(* IEC 61131-3 sources: SafePLC-Gen-Evaluation/Evaluation Results/Dexpi_PDF/run_01, 2 files *)

(* ---- io_declarations.st ---- *)
(* ==================================================  *)
(* PLC I/O Variable Declarations — CODESYS 3.5  *)
(* Generated by SafePLC-Gen Multimodal  *)
(* ==================================================  *)

VAR_GLOBAL
    (* --- Analog Inputs ---  *)
    PI_4712.01_Raw               AT %IW0       : INT := 0;    (* PI-4712.01 — Pressure indicator, local, on process li  *)
    PICSA_4712.02_Raw            AT %IW2       : INT := 0;    (* PICSA-4712.02 — Pressure indicator, controller, switch,   *)
    TICSA_4750.03_Raw            AT %IW4       : INT := 0;    (* TICSA-4750.03 — Temperature indicator, controller, switc  *)
    (* --- Analog Outputs ---  *)
    MV_73KH12_25_Out             AT %QW0       : INT := 0;    (* MV-73KH12-25 — Manual isolation valve on line 73KH12-25  *)
    MV_73KH12_50a_Out            AT %QW2       : INT := 0;    (* MV-73KH12-50a — Manual isolation valve on line 73KH12-50  *)
    MV_73KH12_50b_Out            AT %QW4       : INT := 0;    (* MV-73KH12-50b — Manual isolation valve on line 73KH12-50  *)
    MV_73KH12_50c_Out            AT %QW6       : INT := 0;    (* MV-73KH12-50c — Manual isolation valve on line 73KH12-50  *)
    MV_MNb_47121_Out             AT %QW8       : INT := 0;    (* MV-MNb-47121 — Manual isolation valve on line MNb 47121  *)
    MV_MNb_47122_Out             AT %QW10      : INT := 0;    (* MV-MNb-47122 — Manual isolation valve on line MNb 47122  *)
    MV_MNb_47123_Out             AT %QW12      : INT := 0;    (* MV-MNb-47123 — Manual isolation valve on line MNb 47123  *)
    MV_MNc_47124_Out             AT %QW14      : INT := 0;    (* MV-MNc-47124 — Manual isolation valve on line MNc 47124  *)
    MV_MNc_47125a_Out            AT %QW16      : INT := 0;    (* MV-MNc-47125a — Manual isolation valve on line MNc 47125  *)
    MV_MNc_47125b_Out            AT %QW18      : INT := 0;    (* MV-MNc-47125b — Manual isolation valve on line MNc 47125  *)
    MV_MNc_47126_Out             AT %QW20      : INT := 0;    (* MV-MNc-47126 — Manual isolation valve on line MNc 47126  *)
    MV_MNc_47127_Out             AT %QW22      : INT := 0;    (* MV-MNc-47127 — Manual isolation valve on line MNc 47127  *)
    MV_QSa_47140_Out             AT %QW24      : INT := 0;    (* MV-QSa-47140 — Manual isolation valve on line QSa 47140  *)
    MV_QSb_47141_Out             AT %QW26      : INT := 0;    (* MV-QSb-47141 — Manual isolation valve on line QSb 47141  *)
    MV_WKa_47130_Out             AT %QW28      : INT := 0;    (* MV-WKa-47130 — Manual isolation valve on utility/drain   *)
    MV_WKa_47131_Out             AT %QW30      : INT := 0;    (* MV-WKa-47131 — Manual isolation valve on utility/drain   *)
    PVA_4712.02_Out              AT %QW32      : INT := 0;    (* PVA-4712.02 — Pressure control valve, fail-closed (F.C  *)
    TV_4750.03_Out               AT %QW34      : INT := 0;    (* TV-4750.03 — Temperature control valve, fail-open (F.  *)
    (* --- Digital Inputs ---  *)
    HS_4750.01                   AT %IX0.0     : BOOL := FALSE;    (* HS-4750.01 — Hand switch / operator station (HS), loc  *)
    (* --- Digital Outputs ---  *)
    XV_HS_4750.01                AT %QX0.0     : BOOL := FALSE;    (* XV-HS-4750.01 — Solenoid-operated or pneumatic on/off va  *)
END_VAR

(* ---- generated_code.st ---- *)
(* Generated by SafePLC-Gen Multimodal — CODESYS 3.5 *)
(* IEC 61131-3 Structured Text *)
(* Date: 2026-04-25T13:53:49.815784 *)

PROGRAM PLC_PRG

VAR
    TICSA_4750_03_Raw            AT %IW4       : INT := 0;
    PICSA_4712_02_Raw            AT %IW2       : INT := 0;
    PI_4712_01_Raw               AT %IW0       : INT := 0;
    HS_4750_01                   AT %IX0.0     : BOOL := FALSE;
    TV_4750_03_Out               AT %QW34      : INT := 0;
    PVA_4712_02_Out              AT %QW32      : INT := 0;
    MV_MNb_47121_Out             AT %QW8       : INT := 0;
    MV_MNb_47122_Out             AT %QW10      : INT := 0;
    MV_MNb_47123_Out             AT %QW12      : INT := 0;
    MV_MNc_47124_Out             AT %QW14      : INT := 0;
    MV_MNc_47125a_Out            AT %QW16      : INT := 0;
    MV_MNc_47125b_Out            AT %QW18      : INT := 0;
    MV_MNc_47126_Out             AT %QW20      : INT := 0;
    MV_MNc_47127_Out             AT %QW22      : INT := 0;
    MV_WKa_47130_Out             AT %QW28      : INT := 0;
    MV_WKa_47131_Out             AT %QW30      : INT := 0;
    MV_73KH12_50a_Out            AT %QW2       : INT := 0;
    MV_73KH12_50b_Out            AT %QW4       : INT := 0;
    MV_73KH12_50c_Out            AT %QW6       : INT := 0;
    MV_73KH12_25_Out             AT %QW0       : INT := 0;
    MV_QSa_47140_Out             AT %QW24      : INT := 0;
    MV_QSb_47141_Out             AT %QW26      : INT := 0;
    XV_HS_4750_01                AT %QX0.0     : BOOL := FALSE;
    ESTOP                        AT %IX0.1     : BOOL := FALSE;
    MANUAL_RESET                 AT %IX0.2     : BOOL := FALSE;
END_VAR

VAR
    LOOP_4750_03_TRIP            : BOOL := FALSE;
    LOOP_4712_02_TRIP            : BOOL := FALSE;
    LOOP_104_01_TRIP             : BOOL := FALSE;

    TICSA_4750_03_HH             : BOOL := FALSE;
    TICSA_4750_03_LL             : BOOL := FALSE;
    PICSA_4712_02_HH             : BOOL := FALSE;
    PICSA_4712_02_LL             : BOOL := FALSE;
    SV_104_01_HH                 : BOOL := FALSE;
    SV_104_01_LL                 : BOOL := FALSE;

    SAFE_STATE                   : BOOL := FALSE;
    FirstScan                    : BOOL := TRUE;

    TICSA_4750_03_Scaled         : REAL := 0.0;
    PICSA_4712_02_Scaled         : REAL := 0.0;
    PI_4712_01_Scaled            : REAL := 0.0;

    TICSA_4750_03_HH_SP          : REAL := 180.0;
    TICSA_4750_03_H_SP           : REAL := 160.0;
    TICSA_4750_03_L_SP           : REAL := 20.0;
    TICSA_4750_03_LL_SP          : REAL := 10.0;
    TICSA_4750_03_Deadband       : REAL := 2.0;

    PICSA_4712_02_HH_SP          : REAL := 90.0;
    PICSA_4712_02_H_SP           : REAL := 80.0;
    PICSA_4712_02_L_SP           : REAL := 5.0;
    PICSA_4712_02_LL_SP          : REAL := 2.0;
    PICSA_4712_02_Deadband       : REAL := 1.0;

    PI_4712_01_HH_SP             : REAL := 90.0;
    PI_4712_01_H_SP              : REAL := 80.0;
    PI_4712_01_L_SP              : REAL := 5.0;
    PI_4712_01_LL_SP             : REAL := 2.0;
    PI_4712_01_Deadband          : REAL := 1.0;

    TICSA_4750_03_H              : BOOL := FALSE;
    TICSA_4750_03_L              : BOOL := FALSE;
    TICSA_4750_03_HH_Latch       : SR := (S1 := FALSE, R := FALSE, Q1 := FALSE);
    TICSA_4750_03_LL_Latch       : SR := (S1 := FALSE, R := FALSE, Q1 := FALSE);
    TICSA_4750_03_HH_Ack         : BOOL := FALSE;
    TICSA_4750_03_LL_Ack         : BOOL := FALSE;

    PICSA_4712_02_H              : BOOL := FALSE;
    PICSA_4712_02_L              : BOOL := FALSE;
    PICSA_4712_02_HH_Latch       : SR := (S1 := FALSE, R := FALSE, Q1 := FALSE);
    PICSA_4712_02_LL_Latch       : SR := (S1 := FALSE, R := FALSE, Q1 := FALSE);
    PICSA_4712_02_HH_Ack         : BOOL := FALSE;
    PICSA_4712_02_LL_Ack         : BOOL := FALSE;

    PI_4712_01_H                 : BOOL := FALSE;
    PI_4712_01_L                 : BOOL := FALSE;
    PI_4712_01_HH_Latch          : SR := (S1 := FALSE, R := FALSE, Q1 := FALSE);
    PI_4712_01_LL_Latch          : SR := (S1 := FALSE, R := FALSE, Q1 := FALSE);
    PI_4712_01_HH_Ack            : BOOL := FALSE;
    PI_4712_01_LL_Ack            : BOOL := FALSE;

    TICSA_4750_03_SP             : REAL := 80.0;
    TICSA_4750_03_Kp             : REAL := 1.2;
    TICSA_4750_03_Ki             : REAL := 0.05;
    TICSA_4750_03_Integral       : REAL := 0.0;
    TICSA_4750_03_Error          : REAL := 0.0;
    TICSA_4750_03_Output_Pct     : REAL := 0.0;

    PICSA_4712_02_SP             : REAL := 50.0;
    PICSA_4712_02_Kp             : REAL := 1.0;
    PICSA_4712_02_Ki             : REAL := 0.04;
    PICSA_4712_02_Integral       : REAL := 0.0;
    PICSA_4712_02_Error          : REAL := 0.0;
    PICSA_4712_02_Output_Pct     : REAL := 0.0;

    XV_HS_4750_01_Cmd            : BOOL := FALSE;
    System_Alarm                 : BOOL := FALSE;
END_VAR

IF FirstScan THEN
    LOOP_4750_03_TRIP := TRUE;
    LOOP_4712_02_TRIP := TRUE;
    LOOP_104_01_TRIP  := TRUE;
    SAFE_STATE        := TRUE;
    TV_4750_03_Out    := 32767;
    PVA_4712_02_Out   := 6554;
    MV_MNb_47121_Out  := 6554;
    MV_MNb_47122_Out  := 6554;
    MV_MNb_47123_Out  := 6554;
    MV_MNc_47124_Out  := 6554;
    MV_MNc_47125a_Out := 6554;
    MV_MNc_47125b_Out := 6554;
    MV_MNc_47126_Out  := 6554;
    MV_MNc_47127_Out  := 6554;
    MV_WKa_47130_Out  := 6554;
    MV_WKa_47131_Out  := 6554;
    MV_73KH12_50a_Out := 6554;
    MV_73KH12_50b_Out := 6554;
    MV_73KH12_50c_Out := 6554;
    MV_73KH12_25_Out  := 6554;
    MV_QSa_47140_Out  := 6554;
    MV_QSb_47141_Out  := 6554;
    XV_HS_4750_01     := FALSE;
    FirstScan         := FALSE;
    RETURN;
END_IF;

TICSA_4750_03_Scaled := ((INT_TO_REAL(TICSA_4750_03_Raw) - 6554.0) / (32767.0 - 6554.0)) * 200.0;
PICSA_4712_02_Scaled := ((INT_TO_REAL(PICSA_4712_02_Raw) - 6554.0) / (32767.0 - 6554.0)) * 100.0;
PI_4712_01_Scaled    := ((INT_TO_REAL(PI_4712_01_Raw)    - 6554.0) / (32767.0 - 6554.0)) * 100.0;

IF TICSA_4750_03_Scaled >= TICSA_4750_03_HH_SP THEN
    TICSA_4750_03_HH := TRUE;
ELSIF TICSA_4750_03_Scaled <= (TICSA_4750_03_HH_SP - TICSA_4750_03_Deadband) THEN
    TICSA_4750_03_HH := FALSE;
END_IF;

IF TICSA_4750_03_Scaled >= TICSA_4750_03_H_SP THEN
    TICSA_4750_03_H := TRUE;
ELSIF TICSA_4750_03_Scaled <= (TICSA_4750_03_H_SP - TICSA_4750_03_Deadband) THEN
    TICSA_4750_03_H := FALSE;
END_IF;

IF TICSA_4750_03_Scaled <= TICSA_4750_03_LL_SP THEN
    TICSA_4750_03_LL := TRUE;
ELSIF TICSA_4750_03_Scaled >= (TICSA_4750_03_LL_SP + TICSA_4750_03_Deadband) THEN
    TICSA_4750_03_LL := FALSE;
END_IF;

IF TICSA_4750_03_Scaled <= TICSA_4750_03_L_SP THEN
    TICSA_4750_03_L := TRUE;
ELSIF TICSA_4750_03_Scaled >= (TICSA_4750_03_L_SP + TICSA_4750_03_Deadband) THEN
    TICSA_4750_03_L := FALSE;
END_IF;

TICSA_4750_03_HH_Latch(S1 := TICSA_4750_03_HH,
                        R  := (TICSA_4750_03_HH_Ack AND NOT TICSA_4750_03_HH));
TICSA_4750_03_LL_Latch(S1 := TICSA_4750_03_LL,
                        R  := (TICSA_4750_03_LL_Ack AND NOT TICSA_4750_03_LL));

IF PICSA_4712_02_Scaled >= PICSA_4712_02_HH_SP THEN
    PICSA_4712_02_HH := TRUE;
ELSIF PICSA_4712_02_Scaled <= (PICSA_4712_02_HH_SP - PICSA_4712_02_Deadband) THEN
    PICSA_4712_02_HH := FALSE;
END_IF;

IF PICSA_4712_02_Scaled >= PICSA_4712_02_H_SP THEN
    PICSA_4712_02_H := TRUE;
ELSIF PICSA_4712_02_Scaled <= (PICSA_4712_02_H_SP - PICSA_4712_02_Deadband) THEN
    PICSA_4712_02_H := FALSE;
END_IF;

IF PICSA_4712_02_Scaled <= PICSA_4712_02_LL_SP THEN
    PICSA_4712_02_LL := TRUE;
ELSIF PICSA_4712_02_Scaled >= (PICSA_4712_02_LL_SP + PICSA_4712_02_Deadband) THEN
    PICSA_4712_02_LL := FALSE;
END_IF;

IF PICSA_4712_02_Scaled <= PICSA_4712_02_L_SP THEN
    PICSA_4712_02_L := TRUE;
ELSIF PICSA_4712_02_Scaled >= (PICSA_4712_02_L_SP + PICSA_4712_02_Deadband) THEN
    PICSA_4712_02_L := FALSE;
END_IF;

PICSA_4712_02_HH_Latch(S1 := PICSA_4712_02_HH,
                        R  := (PICSA_4712_02_HH_Ack AND NOT PICSA_4712_02_HH));
PICSA_4712_02_LL_Latch(S1 := PICSA_4712_02_LL,
                        R  := (PICSA_4712_02_LL_Ack AND NOT PICSA_4712_02_LL));

IF PI_4712_01_Scaled >= PI_4712_01_HH_SP THEN
    PI_4712_01_HH_Latch(S1 := TRUE, R := FALSE);
ELSIF PI_4712_01_Scaled <= (PI_4712_01_HH_SP - PI_4712_01_Deadband) THEN
    PI_4712_01_HH_Latch(S1 := FALSE, R := (PI_4712_01_HH_Ack AND NOT (PI_4712_01_Scaled >= PI_4712_01_HH_SP)));
END_IF;

IF PI_4712_01_Scaled >= PI_4712_01_H_SP THEN
    PI_4712_01_H := TRUE;
ELSIF PI_4712_01_Scaled <= (PI_4712_01_H_SP - PI_4712_01_Deadband) THEN
    PI_4712_01_H := FALSE;
END_IF;

IF PI_4712_01_Scaled <= PI_4712_01_LL_SP THEN
    PI_4712_01_LL_Latch(S1 := TRUE, R := FALSE);
ELSIF PI_4712_01_Scaled >= (PI_4712_01_LL_SP + PI_4712_01_Deadband) THEN
    PI_4712_01_LL_Latch(S1 := FALSE, R := (PI_4712_01_LL_Ack AND NOT (PI_4712_01_Scaled <= PI_4712_01_LL_SP)));
END_IF;

IF PI_4712_01_Scaled <= PI_4712_01_L_SP THEN
    PI_4712_01_L := TRUE;
ELSIF PI_4712_01_Scaled >= (PI_4712_01_L_SP + PI_4712_01_Deadband) THEN
    PI_4712_01_L := FALSE;
END_IF;

IF TICSA_4750_03_HH OR TICSA_4750_03_LL THEN
    LOOP_4750_03_TRIP := TRUE;
ELSIF LOOP_4750_03_TRIP AND MANUAL_RESET
      AND NOT TICSA_4750_03_HH AND NOT TICSA_4750_03_LL THEN
    LOOP_4750_03_TRIP := FALSE;
END_IF;

IF PICSA_4712_02_HH OR PICSA_4712_02_LL THEN
    LOOP_4712_02_TRIP := TRUE;
ELSIF LOOP_4712_02_TRIP AND MANUAL_RESET
      AND NOT PICSA_4712_02_HH AND NOT PICSA_4712_02_LL THEN
    LOOP_4712_02_TRIP := FALSE;
END_IF;

IF SV_104_01_HH OR SV_104_01_LL THEN
    LOOP_104_01_TRIP := TRUE;
ELSIF LOOP_104_01_TRIP AND MANUAL_RESET
      AND NOT SV_104_01_HH AND NOT SV_104_01_LL THEN
    LOOP_104_01_TRIP := FALSE;
END_IF;

SAFE_STATE := ESTOP OR LOOP_4750_03_TRIP OR LOOP_4712_02_TRIP OR LOOP_104_01_TRIP;

IF NOT SAFE_STATE THEN
    XV_HS_4750_01_Cmd := HS_4750_01;
    XV_HS_4750_01     := XV_HS_4750_01_Cmd;
ELSE
    XV_HS_4750_01_Cmd := FALSE;
    XV_HS_4750_01     := FALSE;
END_IF;

IF NOT SAFE_STATE THEN
    TICSA_4750_03_Error    := TICSA_4750_03_SP - TICSA_4750_03_Scaled;
    TICSA_4750_03_Integral := TICSA_4750_03_Integral + (TICSA_4750_03_Ki * TICSA_4750_03_Error);
    IF TICSA_4750_03_Integral > 100.0 THEN
        TICSA_4750_03_Integral := 100.0;
    ELSIF TICSA_4750_03_Integral < 0.0 THEN
        TICSA_4750_03_Integral := 0.0;
    END_IF;
    TICSA_4750_03_Output_Pct := (TICSA_4750_03_Kp * TICSA_4750_03_Error) + TICSA_4750_03_Integral;
    IF TICSA_4750_03_Output_Pct > 100.0 THEN
        TICSA_4750_03_Output_Pct := 100.0;
    ELSIF TICSA_4750_03_Output_Pct < 0.0 THEN
        TICSA_4750_03_Output_Pct := 0.0;
    END_IF;
    TV_4750_03_Out := REAL_TO_INT(6554.0 + (TICSA_4750_03_Output_Pct / 100.0) * (32767.0 - 6554.0));
ELSE
    TV_4750_03_Out := 32767;
END_IF;

IF NOT SAFE_STATE THEN
    PICSA_4712_02_Error    := PICSA_4712_02_SP - PICSA_4712_02_Scaled;
    PICSA_4712_02_Integral := PICSA_4712_02_Integral + (PICSA_4712_02_Ki * PICSA_4712_02_Error);
    IF PICSA_4712_02_Integral > 100.0 THEN
        PICSA_4712_02_Integral := 100.0;
    ELSIF PICSA_4712_02_Integral < 0.0 THEN
        PICSA_4712_02_Integral := 0.0;
    END_IF;
    PICSA_4712_02_Output_Pct := (PICSA_4712_02_Kp * PICSA_4712_02_Error) + PICSA_4712_02_Integral;
    IF PICSA_4712_02_Output_Pct > 100.0 THEN
        PICSA_4712_02_Output_Pct := 100.0;
    ELSIF PICSA_4712_02_Output_Pct < 0.0 THEN
        PICSA_4712_02_Output_Pct := 0.0;
    END_IF;
    PVA_4712_02_Out := REAL_TO_INT(6554.0 + (PICSA_4712_02_Output_Pct / 100.0) * (32767.0 - 6554.0));
ELSE
    PVA_4712_02_Out := 6554;
END_IF;

IF SAFE_STATE THEN
    MV_MNb_47121_Out  := 6554;
    MV_MNb_47122_Out  := 6554;
    MV_MNb_47123_Out  := 6554;
    MV_MNc_47124_Out  := 6554;
    MV_MNc_47125a_Out := 6554;
    MV_MNc_47125b_Out := 6554;
    MV_MNc_47126_Out  := 6554;
    MV_MNc_47127_Out  := 6554;
    MV_WKa_47130_Out  := 6554;
    MV_WKa_47131_Out  := 6554;
    MV_73KH12_50a_Out := 6554;
    MV_73KH12_50b_Out := 6554;
    MV_73KH12_50c_Out := 6554;
    MV_73KH12_25_Out  := 6554;
    MV_QSa_47140_Out  := 6554;
    MV_QSb_47141_Out  := 6554;
END_IF;

System_Alarm :=
    TICSA_4750_03_HH_Latch.Q1 OR TICSA_4750_03_LL_Latch.Q1 OR
    TICSA_4750_03_H            OR TICSA_4750_03_L            OR
    PICSA_4712_02_HH_Latch.Q1 OR PICSA_4712_02_LL_Latch.Q1 OR
    PICSA_4712_02_H            OR PICSA_4712_02_L            OR
    PI_4712_01_HH_Latch.Q1    OR PI_4712_01_LL_Latch.Q1    OR
    PI_4712_01_H               OR PI_4712_01_L              OR
    LOOP_4750_03_TRIP          OR LOOP_4712_02_TRIP         OR
    LOOP_104_01_TRIP           OR SAFE_STATE;

END_PROGRAM
